Staubli VAL3: refreshDynamic.pgx

program refreshDynamic()
begin
  // DO NOT CHANGE
  nRefresh=clock()
  use:bUseRefresh=false
  //
  // ADD HERE
  //

 //// call use:type(0,1,"Curr. position : "+toString("",aioGet(io:currentPulse)))


 end
